FUNCTION_BLOCK SampleContext EXTENDS TcoCore.TcoContext
VAR
	_sampleComponent : SampleComponent(THIS^);
END_VAR

(*~
	<docu>
		<summary>
			Main method of the TcoContext. This is the entry point of any control logic that belongs to this context. 
			The call of this method is ensured by calling the <c>InstanceName.Run()</c> method, and it must not be called explicitly.
			This method is abstract, and it must be overridden in derived block.
		</summary>
	</docu>
~*)
METHOD PROTECTED  Main
_sampleComponent.Service();
_sampleComponent();
END_METHOD

END_FUNCTION_BLOCK

(* stored: Version 1.1.0.1, ProductVersion 3.1.4024.9
   POU SampleContext: Id {1f86152d-4972-03a3-3260-0644f5027317}, SpecialFunc None
   Method Main: Id {f6b177a9-ba06-0204-3447-456dc9e8882a} *)
